{attribute 'qualified_only'}
{attribute 'strict'}
TYPE E_Axis_JogMode :
(
	eJogMode_0 := 0,//Kontinuierliche Bewegung
	//eJogMode_1, 	//Tippweg
	eJogMode_1,		//0,01 Tippen
	eJogMode_2,		//0,1 Tippen
	eJogMode_3,		//1 Tippen
	eJogMode_4,		//10 Tippen
	eJogMode_5		//100 Tippen
);
END_TYPE

(* stored: Version 1.1.0.1
   EnumerationTextList E_Axis_JogMode: Id {c9ff2567-0cf2-4265-8697-4bfc1b070e29} *)
